{attribute 'monitoring' := 'variable'}
PROPERTY proAvailable : BOOL
GET
proAvailable := proIsReady;
END_GET
END_PROPERTY

{attribute 'monitoring' := 'variable'}
PROPERTY proLockDown : BOOL
GET
proLockDown := proIsError;
END_GET
END_PROPERTY

END_FUNCTION_BLOCK

// 21 Interface/ITF_SPERRANTRIEB
INTERFACE ITF_SPERRANTRIEB EXTENDS CtaAppBmk.ITF_BMK, CtaAppModbusSpezifikation.ITF_MODBUS_SPEZIFIKATION

PROPERTY proAuto : BOOL
GET
END_GET
SET
END_SET
END_PROPERTY

PROPERTY proHandOff : BOOL
GET
END_GET
SET
END_SET
END_PROPERTY

PROPERTY proHandOn : BOOL
GET
END_GET
SET
END_SET
END_PROPERTY

PROPERTY proIsRegulatet : BOOL
GET
END_GET
END_PROPERTY

PROPERTY proIsError : BOOL
GET
END_GET
END_PROPERTY

PROPERTY proIsWarning : BOOL
GET
END_GET
END_PROPERTY

PROPERTY proIsEnabled : BOOL
GET
END_GET
END_PROPERTY

PROPERTY proIsHandOnOrOff : BOOL
GET
END_GET
END_PROPERTY

PROPERTY proIsReady : BOOL
GET
END_GET
END_PROPERTY

PROPERTY proHardWareHandModulAktive : BOOL
GET
END_GET
END_PROPERTY

PROPERTY proRevisionSwitchOk : BOOL
GET
END_GET
END_PROPERTY

PROPERTY proHandManualClose : BOOL
SET
END_SET
GET
END_GET
END_PROPERTY

PROPERTY proEn : BOOL
SET
END_SET
GET
END_GET
END_PROPERTY

PROPERTY proRükIsOpen : BOOL
GET
END_GET
END_PROPERTY

PROPERTY proRükIsClosed : BOOL
GET
END_GET
END_PROPERTY

PROPERTY INTERNAL proStateSymbol : STRING
GET
END_GET
END_PROPERTY

PROPERTY INTERNAL proEnSymbol : STRING
GET
END_GET
END_PROPERTY

PROPERTY proOnZu : BOOL
GET
END_GET
END_PROPERTY

PROPERTY proIsOnY : REAL
GET
END_GET
END_PROPERTY

PROPERTY proOnAuf : BOOL
GET
END_GET
END_PROPERTY

PROPERTY proOnY : REAL
GET
END_GET
END_PROPERTY

PROPERTY proGetDI_RükIsOpen : BOOL
GET
END_GET
END_PROPERTY

PROPERTY proNotShowDI_RükIsOpen : BOOL
GET
END_GET
END_PROPERTY

PROPERTY proIsOpen_ITF : CtaSysIO.ITF_IO
GET
END_GET
END_PROPERTY

PROPERTY INTERNAL proGetDI_ActuatorHand : BOOL
GET
END_GET
END_PROPERTY

PROPERTY proNotShowDI_ActuatorHand : BOOL
GET
END_GET
END_PROPERTY

PROPERTY proHandModul_ITF : CtaSysIO.ITF_IO
GET
END_GET
END_PROPERTY

PROPERTY INTERNAL proGetDI_ActuatorFuseOk : BOOL
GET
END_GET
END_PROPERTY

PROPERTY proNotShowDI_ActuatorFuseOk : BOOL
GET
END_GET
END_PROPERTY

PROPERTY proActuatorFuse_ITF : CtaSysIO.ITF_IO
GET
END_GET
END_PROPERTY

PROPERTY INTERNAL proGetDI_IsReady : BOOL
GET
END_GET
END_PROPERTY

PROPERTY proNotShowDI_Ready : BOOL
GET
END_GET
END_PROPERTY

PROPERTY proActuatorReady_ITF : CtaSysIO.ITF_IO
GET
END_GET
END_PROPERTY

PROPERTY INTERNAL proGetDI_FuseOK : BOOL
GET
END_GET
END_PROPERTY

PROPERTY proNotShowDI_FuseOk : BOOL
GET
END_GET
END_PROPERTY

PROPERTY proFuse_ITF : CtaSysIO.ITF_IO
GET
END_GET
END_PROPERTY

PROPERTY INTERNAL proGetDI_RevisionSwitchOK : BOOL
GET
END_GET
END_PROPERTY

PROPERTY proNotShowDI_RevisionSwitchOk : BOOL
GET
END_GET
END_PROPERTY

PROPERTY proRevisionSwitch_ITF : CtaSysIO.ITF_IO
GET
END_GET
END_PROPERTY

PROPERTY proNotShowAI_ActualPosition : BOOL
GET
END_GET
END_PROPERTY

PROPERTY proGetAI_ActualPosition : REAL
GET
END_GET
END_PROPERTY

PROPERTY proActualPosition_ITF : CtaSysIO.ITF_IO
GET
END_GET
END_PROPERTY

PROPERTY proGetDI_RükIsClosed : BOOL
GET
END_GET
END_PROPERTY

PROPERTY proNotShowDI_RükIsClosed : BOOL
GET
END_GET
END_PROPERTY

PROPERTY proIsClosed_ITF : CtaSysIO.ITF_IO
GET
END_GET
END_PROPERTY

PROPERTY proOnY_ITF : CtaSysIO.ITF_IO
GET
END_GET
END_PROPERTY

PROPERTY proOnOpen_ITF : CtaSysIO.ITF_IO
GET
END_GET
END_PROPERTY

PROPERTY proOnClose_ITF : CtaSysIO.ITF_IO
GET
END_GET
END_PROPERTY

PROPERTY INTERNAL proAnzWarning : INT
GET
END_GET
END_PROPERTY

PROPERTY INTERNAL proITF_REPORTMANAGER : CtaAppReport.ITF_REPORTMANAGER
GET
END_GET
END_PROPERTY

PROPERTY INTERNAL proAnzInfo : INT
GET
END_GET
END_PROPERTY

PROPERTY INTERNAL proAnzError : INT
GET
END_GET
END_PROPERTY

PROPERTY INTERNAL proModbusTest : BOOL
SET
END_SET
GET
END_GET
END_PROPERTY

PROPERTY proModbusStateWord : REFERENCE TO ARRAY[0..3] OF WORD
GET
END_GET
END_PROPERTY

PROPERTY proModbusControllWord : REFERENCE TO ARRAY[0..3] OF WORD
GET
END_GET
END_PROPERTY

PROPERTY proConfigError : BOOL
GET
END_GET
END_PROPERTY

PROPERTY p_scBase_fbxEnable : CtaSysConfig.ITF_DATATYPE;
GET
END_GET
END_PROPERTY

PROPERTY p_scBase_fbxControllMb : CtaSysConfig.ITF_DATATYPE;
GET
END_GET
END_PROPERTY

PROPERTY p_scBase_fbxInvertiert : CtaSysConfig.ITF_DATATYPE;
GET
END_GET
END_PROPERTY

PROPERTY p_scBase_fbtSettingTime : CtaSysConfig.ITF_DATATYPE;
GET
END_GET
END_PROPERTY

PROPERTY p_scFuse_fbxEnable : CtaSysConfig.ITF_DATATYPE;
GET
END_GET
END_PROPERTY

PROPERTY p_scFuse_fbxInputMb : CtaSysConfig.ITF_DATATYPE;
GET
END_GET
END_PROPERTY

PROPERTY p_scFuse_fbxDoesAlarm : CtaSysConfig.ITF_DATATYPE;
GET
END_GET
END_PROPERTY

PROPERTY p_scActuatorFuse_fbxEnable : CtaSysConfig.ITF_DATATYPE;
GET
END_GET
END_PROPERTY

PROPERTY p_scActuatorFuse_fbxInputMb : CtaSysConfig.ITF_DATATYPE;
GET
END_GET
END_PROPERTY

PROPERTY p_scActuatorFuse_fbxDoesAlarm : CtaSysConfig.ITF_DATATYPE;
GET
END_GET
END_PROPERTY

PROPERTY p_scInSperrAtRevisionSwitch_fbxEnable : CtaSysConfig.ITF_DATATYPE;
GET
END_GET
END_PROPERTY

PROPERTY p_scInSperrAtRevisionSwitch_fbxInputMb : CtaSysConfig.ITF_DATATYPE;
GET
END_GET
END_PROPERTY

PROPERTY p_scInSperrAtReady_fbxEnable : CtaSysConfig.ITF_DATATYPE;
GET
END_GET
END_PROPERTY

PROPERTY p_scInSperrAtReady_fbxInputMb : CtaSysConfig.ITF_DATATYPE;
GET
END_GET
END_PROPERTY

PROPERTY p_scInSperrAtHand_fbxEnable : CtaSysConfig.ITF_DATATYPE;
GET
END_GET
END_PROPERTY

PROPERTY p_scInSperrAtHand_fbxInputMb : CtaSysConfig.ITF_DATATYPE;
GET
END_GET
END_PROPERTY

PROPERTY p_scInSperrAtRükClosed_fbxEnable : CtaSysConfig.ITF_DATATYPE;
GET
END_GET
END_PROPERTY

PROPERTY p_scInSperrAtRükClosed_fbxInputMb : CtaSysConfig.ITF_DATATYPE;
GET
END_GET
END_PROPERTY

PROPERTY p_scInSperrAtRükClosed_fbxDoesAlarm : CtaSysConfig.ITF_DATATYPE;
GET
END_GET
END_PROPERTY

PROPERTY p_scInSperrAtRükClosed_fbtDelayStart : CtaSysConfig.ITF_DATATYPE;
GET
END_GET
END_PROPERTY

PROPERTY p_scInSperrAtRükClosed_fbtDelayRun : CtaSysConfig.ITF_DATATYPE;
GET
END_GET
END_PROPERTY

PROPERTY p_scInSperrAtRükClosed_fbiTypeOfAck : CtaSysConfig.ITF_DATATYPE;
GET
END_GET
END_PROPERTY

PROPERTY p_scInSperrAtRükClosed_fbiMaxErrorRetryAllowed : CtaSysConfig.ITF_DATATYPE;
GET
END_GET
END_PROPERTY

PROPERTY p_scInSperrAtRükOpen_fbxEnable : CtaSysConfig.ITF_DATATYPE;
GET
END_GET
END_PROPERTY

PROPERTY p_scInSperrAtRükOpen_fbxInputMb : CtaSysConfig.ITF_DATATYPE;
GET
END_GET
END_PROPERTY

PROPERTY p_scInSperrAtRükOpen_fbxDoesAlarm : CtaSysConfig.ITF_DATATYPE;
GET
END_GET
END_PROPERTY

PROPERTY p_scInSperrAtRükOpen_fbtDelayStart : CtaSysConfig.ITF_DATATYPE;
GET
END_GET
END_PROPERTY

PROPERTY p_scInSperrAtRükOpen_fbtDelayRun : CtaSysConfig.ITF_DATATYPE;
GET
END_GET
END_PROPERTY

PROPERTY p_scInSperrAtRükOpen_fbiTypeOfAck : CtaSysConfig.ITF_DATATYPE;
GET
END_GET
END_PROPERTY

PROPERTY p_scInSperrAtRükOpen_fbiMaxErrorRetryAllowed : CtaSysConfig.ITF_DATATYPE;
GET
END_GET
END_PROPERTY

PROPERTY p_scInSperrAtActualPosition_fbxEnable : CtaSysConfig.ITF_DATATYPE;
GET
END_GET
END_PROPERTY

PROPERTY p_scInSperrAtActualPosition_fbxInputMb : CtaSysConfig.ITF_DATATYPE;
GET
END_GET
END_PROPERTY

PROPERTY p_scInSperrAtActualPosition_fbxDoesAlarm : CtaSysConfig.ITF_DATATYPE;
GET
END_GET
END_PROPERTY

PROPERTY p_scInSperrAtActualPosition_fbrMaxDiff : CtaSysConfig.ITF_DATATYPE;
GET
END_GET
END_PROPERTY

PROPERTY p_scInSperrAtActualPosition_fbtDelayStart : CtaSysConfig.ITF_DATATYPE;
GET
END_GET
END_PROPERTY

PROPERTY p_scInSperrAtActualPosition_fbtDelayRun : CtaSysConfig.ITF_DATATYPE;
GET
END_GET
END_PROPERTY

PROPERTY p_scInSperrAtActualPosition_fbiTypeOfAck : CtaSysConfig.ITF_DATATYPE;
GET
END_GET
END_PROPERTY

PROPERTY p_scInSperrAtActualPosition_fbiMaxErrorRetryAllowed : CtaSysConfig.ITF_DATATYPE;
GET
END_GET
END_PROPERTY

PROPERTY p_scInfluxDb_fbxEnable : CtaSysConfig.ITF_DATATYPE;
GET
END_GET
END_PROPERTY

PROPERTY p_scManual_fbxAlowManualOn : CtaSysConfig.ITF_DATATYPE;
GET
END_GET
END_PROPERTY

PROPERTY p_scManual_fbuiManualState : CtaSysConfig.ITF_DATATYPE;
GET
END_GET
END_PROPERTY

PROPERTY p_scManual_fbuiSchaltBefehl : CtaSysConfig.ITF_DATATYPE;
GET
END_GET
END_PROPERTY

PROPERTY proHandManualOpen : BOOL
GET
END_GET
SET
END_SET
END_PROPERTY

PROPERTY proIsInverted : BOOL
GET
END_GET
END_PROPERTY

PROPERTY proKlappenStatus : enKlappenStatus
GET
END_GET
END_PROPERTY

PROPERTY proValveIcon : UINT
GET
END_GET
SET
END_SET
END_PROPERTY

{attribute 'monitoring' := 'variable'}
PROPERTY proAcknowlege : BOOL
GET
END_GET
END_PROPERTY

{attribute 'monitoring' := 'variable'}
PROPERTY proAvailable : BOOL
GET
END_GET
END_PROPERTY

{attribute 'monitoring' := 'variable'}
PROPERTY proLockDown : BOOL
GET
END_GET
END_PROPERTY

PROPERTY proOn : BOOL
GET
END_GET
END_PROPERTY

END_INTERFACE

// 30 Program Organization Units/fcGetBigerStringValue
FUNCTION fcGetBigerStringValue : INT
VAR_INPUT
    st1     :   STRING(255);
    st2     :   STRING(255);
END_VAR
VAR
    diFor: DINT;
    diMax: DINT;
END_VAR

IF LEN(st1) > LEN(st2) THEN
    diMax := LEN(st2); 
    fcGetBigerStringValue := 1;
ELSIF LEN(st1) < LEN(st2) THEN
    diMax := LEN(st1);
    fcGetBigerStringValue := 2;     
ELSE
    diMax := LEN(st1);    
END_IF;
FOR diFor := 0 TO  diMax DO
    IF st1[diFor] > st2[diFor] THEN
        fcGetBigerStringValue := 1;  
        EXIT; 
    ELSIF st1[diFor] < st2[diFor] THEN
        fcGetBigerStringValue := 2;  
        EXIT;
    END_IF;
END_FOR;

END_FUNCTION

// 30 Program Organization Units/fcCheckQuerryReturnIcon
FUNCTION fcCheckQuerryReturnIcon : BOOL
VAR_INPUT
	_ITF_In			:	ITF_SPERRANTRIEB;
	_uiIconNr_In	:	UINT;
END_VAR

IF __QUERYINTERFACE(_ITF_In,_ITF_In) THEN	
	fcCheckQuerryReturnIcon := TRUE;	
	_ITF_In.proValveIcon := _uiIconNr_In;
ELSE
	fcCheckQuerryReturnIcon := FALSE;	
END_IF

END_FUNCTION

// 40 Visualizations/POPUP/SperrAntrieb_POPUP
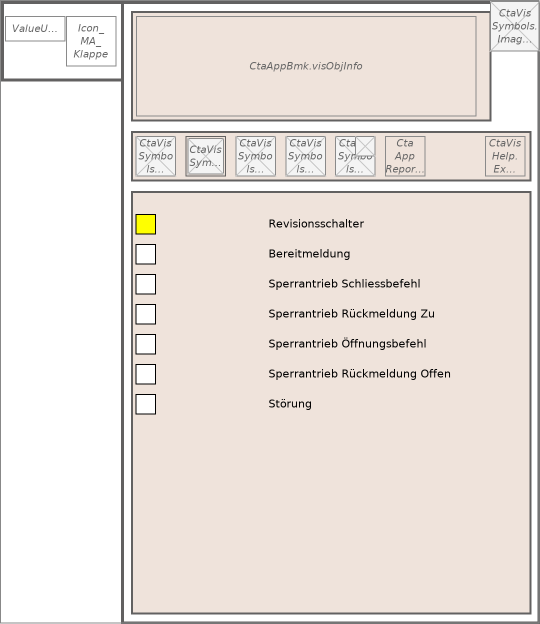
VISUALIZATION SperrAntrieb_POPUP  // 540x624
VAR_INPUT
    ITF_SPERRANTRIEBIN  :   ITF_SPERRANTRIEB;
    stExklParameter		:   STRING[40];	
	uiPopUpGruppe		: UINT;
END_VAR
    RoundedRectangle (1,1 160x80)
    RoundedRectangle (121,1 419x623)
    RoundedRectangle (131,11 360x110)
    RoundedRectangle (131,191 400x423)
    RoundedRectangle (131,131 400x50)
    Frame (136,16 340x100)
        shows CtaAppBmk.visObjInfo(ITF_BMK_IN := ITF_SPERRANTRIEBIN)
    Image (490,1 50x50), image: CtaVisSymbols.ImagePool.close_solo_black
        OnMouseClick:  Dialog=SperrAntrieb_POPUP, Result=None, NumpadKeypadSet=True
    Frame (131,204 399x400), frame switch variable: uiPopUpGruppe
        shows SperrAntrieb_OVERVIEW(ITF_SPERRANTRIEBIN := ITF_SPERRANTRIEBIN)
        shows SperrAntrieb_MANUAL(ITF_SPERRANTRIEBIN := ITF_SPERRANTRIEBIN)
        shows SperrAntrieb_PARAMETER(ITF_SPERRANTRIEBIN := ITF_SPERRANTRIEBIN)
        shows SperrAntrieb_IO(ITF_SPERRANTRIEBIN := ITF_SPERRANTRIEBIN)
        shows SperrAntrieb_BUS(ITF_SPERRANTRIEBIN := ITF_SPERRANTRIEBIN)
        shows SperrAntrieb_REPORTS(ITF_SPERRANTRIEBIN := ITF_SPERRANTRIEBIN)
        pReferences[2]: ITF_Parameter=ITF_SPERRANTRIEBIN.proParameter
    Frame (131,136 399x40)
        shows SperrAntrieb_PopUpListe(uiPopUpGruppe := uiPopUpGruppe, xHand := ITF_SPERRANTRIEBIN.proIsHandOnOrOff, xHandOff := ITF_SPERRANTRIEBIN.proHandOff, ITF_REPORTMANAGER_IN := ITF_SPERRANTRIEBIN.proITF_REPORTMANAGER, xBusTestAktiv := ITF_SPERRANTRIEBIN.proModbusTest, stExklParameter_IN := stExklParameter)
        pReferences[0]: AnzError=ITF_SPERRANTRIEBIN.proAnzError, AnzWarning=ITF_SPERRANTRIEBIN.proAnzWarning
    Frame (5,16 110x50), input disabled if: TRUE, frame switch variable: ITF_SPERRANTRIEBIN.proValveIcon
        shows SperrAntrieb_MA_Flap_Txt_L_Above(ITF_SPERRANTRIEB_IN := ITF_SPERRANTRIEBIN, stExklParameter := stExklParameter)
        shows SperrAntrieb_MB_Flap_Txt_L_Below(ITF_SPERRANTRIEB_IN := ITF_SPERRANTRIEBIN, stExklParameter := stExklParameter)
        shows SperrAntrieb_ML_Flap_Txt_L_Above(ITF_SPERRANTRIEB_IN := ITF_SPERRANTRIEBIN, stExklParameter := stExklParameter)
        shows SperrAntrieb_ML_Flap_Txt_L_Below(ITF_SPERRANTRIEB_IN := ITF_SPERRANTRIEBIN, stExklParameter := stExklParameter)
        shows SperrAntrieb_MA_Flap_Txt_R_Above(ITF_SPERRANTRIEB_IN := ITF_SPERRANTRIEBIN, stExklParameter := stExklParameter)
        shows SperrAntrieb_MB_Flap_Right_Txt_R_Below(ITF_SPERRANTRIEB_IN := ITF_SPERRANTRIEBIN, stExklParameter := stExklParameter)
        shows SperrAntrieb_MR_Flap_Txt_R_Above(ITF_SPERRANTRIEB_IN := ITF_SPERRANTRIEBIN, stExklParameter := stExklParameter)
        shows SperrAntrieb_MR_Flap_Txt_R_Below(ITF_SPERRANTRIEB_IN := ITF_SPERRANTRIEBIN, stExklParameter := stExklParameter)
        shows S_AT_ML_Valve_AB_Down_Txt_L_Above(ITF_STELLANTRIEB_IN := ITF_STELLANTRIEBIN)
        shows S_AT_ML_Valve_AB_Down_Txt_L_Below(ITF_STELLANTRIEB_IN := ITF_STELLANTRIEBIN)
        shows S_AT_ML_Valve_AB_Up_Txt_L_Above(ITF_STELLANTRIEB_IN := ITF_STELLANTRIEBIN)
        shows S_AT_ML_Valve_AB_Up_Txt_L_Below(ITF_STELLANTRIEB_IN := ITF_STELLANTRIEBIN)
        shows S_AT_ML_Valve_Flow_Txt_L_Above(ITF_STELLANTRIEB_IN := ITF_STELLANTRIEBIN)
        shows S_AT_ML_Valve_Flow_Txt_L_Below(ITF_STELLANTRIEB_IN := ITF_STELLANTRIEBIN)
        shows S_AT_ML_Valve_Mix_Txt_L_Above(ITF_STELLANTRIEB_IN := ITF_STELLANTRIEBIN)
        shows S_AT_ML_Valve_Mix_Txt_L_Below(ITF_STELLANTRIEB_IN := ITF_STELLANTRIEBIN)
        shows S_AT_MA_Valve_AB_Left_Txt_R_Above(ITF_STELLANTRIEB_IN := ITF_STELLANTRIEBIN)
        shows S_AT_MA_Valve_AB_Right_Txt_R_Above(ITF_STELLANTRIEB_IN := ITF_STELLANTRIEBIN)
        shows S_AT_MA_Valve_Flow_Txt_R_Above(ITF_STELLANTRIEB_IN := ITF_STELLANTRIEBIN)
        shows S_AT_MA_Valve_Mix_Txt_R_Above(ITF_STELLANTRIEB_IN := ITF_STELLANTRIEBIN)
        shows S_AT_MB_Valve_AB_Left_Txt_R_Below(ITF_STELLANTRIEB_IN := ITF_STELLANTRIEBIN)
        shows S_AT_MB_Valve_AB_Right_Txt_R_Below(ITF_STELLANTRIEB_IN := ITF_STELLANTRIEBIN)
        shows S_AT_MB_Valve_Flow_Txt_R_Below(ITF_STELLANTRIEB_IN := ITF_STELLANTRIEBIN)
        shows S_AT_MB_Valve_Mix_Txt_R_Below(ITF_STELLANTRIEB_IN := ITF_STELLANTRIEBIN)
        shows S_AT_MR_Valve_AB_Down_Txt_R_Above(ITF_STELLANTRIEB_IN := ITF_STELLANTRIEBIN)
        shows S_AT_MR_Valve_AB_Down_Txt_R_Below(ITF_STELLANTRIEB_IN := ITF_STELLANTRIEBIN)
        shows S_AT_MR_Valve_AB_Up_Txt_R_Above(ITF_STELLANTRIEB_IN := ITF_STELLANTRIEBIN)
        shows S_AT_MR_Valve_AB_Up_Txt_R_Below(ITF_STELLANTRIEB_IN := ITF_STELLANTRIEBIN)
        shows S_AT_MR_Valve_Flow_Txt_R_Above(ITF_STELLANTRIEB_IN := ITF_STELLANTRIEBIN)
        shows S_AT_MR_Valve_Flow_Txt_R_Below(ITF_STELLANTRIEB_IN := ITF_STELLANTRIEBIN)
        shows S_AT_MR_Valve_Mix_Txt_R_Above(ITF_STELLANTRIEB_IN := ITF_STELLANTRIEBIN)
        shows S_AT_MR_Valve_Mix_Txt_R_Below(ITF_STELLANTRIEB_IN := ITF_STELLANTRIEBIN)
        shows S_AT_MR_Valve_AB_Up_Txt_R_Above()
        shows S_AT_MR_Valve_AB_Up_Txt_R_Below()
        shows S_AT_MR_Flap_Txt_R_Above()
        shows S_AT_MR_Flap_Txt_R_Below()
        shows S_AT_MR_Valve_Flow_Txt_R_Above()
        shows S_AT_MR_Valve_Flow_Txt_R_Below()
        shows S_AT_MR_Valve_Mix_Txt_R_Above()
        shows S_AT_MR_Valve_Mix_Txt_R_Below()
END_VISUALIZATION

// 40 Visualizations/POPUP/SperrAntrieb_PopUpListe
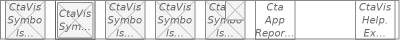
VISUALIZATION SperrAntrieb_PopUpListe  // 400x40
VAR_IN_OUT
	uiPopUpGruppe 			:	UINT;
END_VAR
VAR_INPUT
    xHand           		: 	BOOL;
    xHandOff        		: 	BOOL;
    ITF_REPORTMANAGER_IN 	: 	CtaAppReport.ITF_REPORTMANAGER;
    xBusTestAktiv   		: 	BOOL;	
	stExklParameter_IN		:	STRING[40];
END_VAR
    Group (5,0 40x40)
        RoundedRectangle (0,0 40x40), colour toggle: uiPopUpGruppe = 0
            OnMouseDown: execute { uiPopUpGruppe := 0; }
        Image (0,0 40x40), image: CtaVisSymbols.ImagePool.eye
            OnMouseDown: execute { uiPopUpGruppe := 0; }
    Group (105,0 40x40)
        RoundedRectangle (0,0 40x40), colour toggle: uiPopUpGruppe = 2
            OnMouseDown: execute { uiPopUpGruppe := 2; }
        Image (0,0 40x40), image: CtaVisSymbols.ImagePool.gear
            OnMouseDown: execute { uiPopUpGruppe := 2; }
    Group (55,0 40x40)
        RoundedRectangle (0,0 40x40), colour toggle: uiPopUpGruppe = 1
            OnMouseDown: execute { uiPopUpGruppe := 1; }
        Image (2,2 36x36), image: CtaVisSymbols.ImagePool.front_hand_Black
            OnMouseDown: execute { uiPopUpGruppe := 1; }
        Image (2,2 36x36), invisible if: NOT xHand, image: CtaVisSymbols.ImagePool.front_hand_Yellow
            OnMouseDown: execute { uiPopUpGruppe := 1; }
        Image (2,2 36x36), invisible if: NOT xHandOff, image: CtaVisSymbols.ImagePool.front_hand_Yellow_Off
            OnMouseDown: execute { uiPopUpGruppe := 1; }
    Group (155,0 40x40)
        RoundedRectangle (0,0 40x40), colour toggle: uiPopUpGruppe = 3
            OnMouseDown: execute { uiPopUpGruppe := 3; }
        Image (0,0 40x40), image: CtaVisSymbols.ImagePool.dip-switch
            OnMouseDown: execute { uiPopUpGruppe := 3; }
    Group (205,0 40x40)
        RoundedRectangle (0,0 40x40), colour toggle: uiPopUpGruppe = 4
            OnMouseDown: execute { uiPopUpGruppe := 4; }
        Image (0,0 40x40), image: CtaVisSymbols.ImagePool.lan
            OnMouseDown: execute { uiPopUpGruppe := 4; }
        Image (20,0 20x20), invisible if: NOT xBusTestAktiv, image: CtaVisSymbols.ImagePool.front_hand_Yellow
            OnMouseDown: execute { uiPopUpGruppe := 4; }
    Group (255,0 40x40)
        RoundedRectangle (0,0 40x40), colour toggle: uiPopUpGruppe = 5
            OnMouseDown: execute { uiPopUpGruppe := 5; }
        Frame (0,0 40x40), input disabled if: TRUE
            shows CtaAppReport.VIS_ANZ_REPORTS_MODUL(ITF_REPORTMANAGER_IN := ITF_REPORTMANAGER_IN)
            OnMouseDown: execute { uiPopUpGruppe := 5; }
    Group (355,0 40x40)
        RoundedRectangle (0,0 40x40), invisible if: stExklParameter_IN = ' '
        Frame (0,0 40x40)
            shows CtaVisHelp.ExkParameterSymbol(stExklParameter := stExklParameter_IN)
END_VISUALIZATION

// 40 Visualizations/ICON/SperrAntrieb_BASE/Icons/Motor
VISUALIZATION Motor  // 15x15
VAR_INPUT
    ITF_SPERRANTRIEB_IN   :   ITF_SPERRANTRIEB;	
END_VAR
    Ellipse (0,0 15x15), "M", colour toggle: ITF_SPERRANTRIEB_IN.proIsError
    Ellipse (0,0 15x15), "M", colour toggle: ITF_SPERRANTRIEB_IN.proOn, invisible if: ITF_SPERRANTRIEB_IN.proIsError
END_VISUALIZATION

// 40 Visualizations/POPUP/PARAMETER/SperrAntrieb_PARAMETER
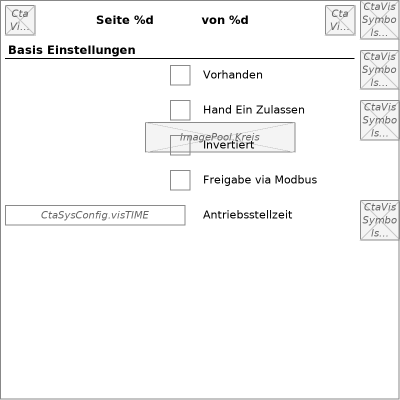
VISUALIZATION SperrAntrieb_PARAMETER  // 400x400
VAR_INPUT
    ITF_SPERRANTRIEBIN : ITF_SPERRANTRIEB;
END_VAR
VAR
    uiParameterGruppe : UINT;
END_VAR
    Image (145,122 150x30), image: ImagePool.Kreis
    Frame (360,0 40x300)
        shows SperrAntrieb_ParameterListe(uiParameterGruppe := uiParameterGruppe)
    Frame (0,0 360x400), frame switch variable: uiParameterGruppe
        shows SperrAntrieb_ParameterBase(ITF_SPERRANTRIEBIN := ITF_SPERRANTRIEBIN)
        shows SperrAntrieb_ParameterFuses(ITF_SPERRANTRIEBIN := ITF_SPERRANTRIEBIN)
        shows SperrAntrieb_ParameterIO(ITF_SPERRANTRIEBIN := ITF_SPERRANTRIEBIN)
        shows SperrAntrieb_ParameterInfluxDb(ITF_SPERRANTRIEBIN := ITF_SPERRANTRIEBIN)
        shows S_AT_ParameterInfluxDb(ITF_Parameter := ITF_Parameter)
        pReferences[0]: ITF_Parameter=ITF_Parameter
        pReferences[1]: ITF_Parameter=ITF_Parameter
        pReferences[2]: ITF_Parameter=ITF_Parameter
        pReferences[3]: ITF_Parameter=ITF_Parameter
END_VISUALIZATION

// 40 Visualizations/POPUP/PARAMETER/SperrAntrieb_ParameterListe
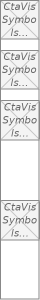
VISUALIZATION SperrAntrieb_ParameterListe  // 40x300
VAR_IN_OUT
	uiParameterGruppe : UINT;
END_VAR
    RoundedRectangle (0,100 39x39), colour toggle: uiParameterGruppe = 2
        OnMouseDown: execute { uiParameterGruppe := 2; }
    RoundedRectangle (0,50 39x39), colour toggle: uiParameterGruppe = 1
        OnMouseDown: execute { uiParameterGruppe := 1; }
    RoundedRectangle (0,0 39x39), colour toggle: uiParameterGruppe = 0
        OnMouseDown: execute { uiParameterGruppe := 0; }
    RoundedRectangle (0,200 39x39), colour toggle: uiParameterGruppe = 3
        OnMouseDown: execute { uiParameterGruppe := 3; }
    Image (0,0 39x39), image: CtaVisSymbols.ImagePool.valve_24dp_000000_FILL0_wght400_GRAD0_opsz24
        OnMouseDown: execute { uiParameterGruppe := 0; }
    Image (0,50 39x39), image: CtaVisSymbols.ImagePool.electric_bolt_24dp_000000_FILL0_wght400_GRAD0_opsz24
        OnMouseDown: execute { uiParameterGruppe := 1; }
    Image (0,100 40x40), image: CtaVisSymbols.ImagePool.dip-switch
        OnMouseDown: execute { uiParameterGruppe := 2; }
    Image (0,200 40x40), image: CtaVisSymbols.ImagePool.sine-wave
        OnMouseDown: execute { uiParameterGruppe := 3; }
END_VISUALIZATION

// 40 Visualizations/POPUP/MANUAL/SperrAntrieb_MANUAL
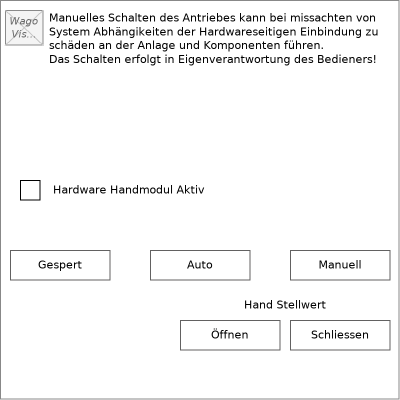
VISUALIZATION SperrAntrieb_MANUAL  // 400x400
VAR_INPUT
    ITF_SPERRANTRIEBIN    :   ITF_SPERRANTRIEB;	
END_VAR
    Label (46,10 350x100), "Manuelles Schalten des Antriebes kann bei missachten von System Abhängikeiten der Hardwareseitigen Einbindung zu schäden an der Anlage und Komponenten führen. Das Schalten erfolgt in Eigenverantwortung des Bedieners!"
    Image (5,10 38x35), image: WagoVisuIcons.WagoIcons.2
    Label (235,295 100x20), "Hand Stellwert"
    Rectangle (20,180 20x20), colour toggle: ITF_SPERRANTRIEBIN.proHardWareHandModulAktive, invisible if: NOT ITF_SPERRANTRIEBIN.proHardWareHandModulAktive
    Label (50,180 200x20), "Hardware Handmodul Aktiv", invisible if: NOT ITF_SPERRANTRIEBIN.proHardWareHandModulAktive
    RoundedRectangle (10,250 100x30), "Gespert", colour toggle: ITF_SPERRANTRIEBIN.proHandOff
        toggle ITF_SPERRANTRIEBIN.proHandOff
    RoundedRectangle (150,250 100x30), "Auto", colour toggle: ITF_SPERRANTRIEBIN.proAuto
        toggle ITF_SPERRANTRIEBIN.proAuto
    RoundedRectangle (290,250 100x30), "Manuell", colour toggle: ITF_SPERRANTRIEBIN.proHandOn
        toggle ITF_SPERRANTRIEBIN.proHandOn
    RoundedRectangle (180,320 100x30), "Öffnen", colour toggle: ITF_SPERRANTRIEBIN.proHandManualOpen, invisible if: NOT ITF_SPERRANTRIEBIN.proHandOn
        toggle ITF_SPERRANTRIEBIN.proHandManualOpen
    RoundedRectangle (290,320 100x30), "Schliessen", colour toggle: ITF_SPERRANTRIEBIN.proHandManualClose, invisible if: NOT ITF_SPERRANTRIEBIN.proHandOn
        toggle ITF_SPERRANTRIEBIN.proHandManualClose
END_VISUALIZATION

// 40 Visualizations/POPUP/OVERVIEW/SperrAntrieb_OVERVIEW
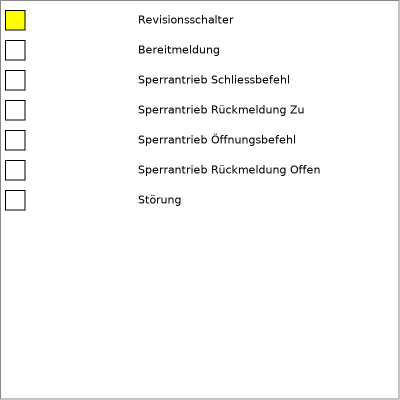
VISUALIZATION SperrAntrieb_OVERVIEW  // 400x400
VAR_INPUT
    ITF_SPERRANTRIEBIN    :   ITF_SPERRANTRIEB;	
END_VAR
    Label (135,10 250x20), "Revisionsschalter"
    Label (135,40 250x20), "Bereitmeldung"
    Rectangle (5,10 20x20), colour toggle: ITF_SPERRANTRIEBIN.proRevisionSwitchOk
    Rectangle (5,40 20x20), colour toggle: ITF_SPERRANTRIEBIN.proIsReady
    Rectangle (5,70 20x20), colour toggle: ITF_SPERRANTRIEBIN.proOnZu
    Label (135,70 250x20), "Sperrantrieb Schliessbefehl"
    Rectangle (5,100 20x20), colour toggle: ITF_SPERRANTRIEBIN.proRükIsClosed, invisible if: ITF_SPERRANTRIEBIN.proNotShowDI_RükIsClosed
    Label (135,100 250x20), "Sperrantrieb Rückmeldung Zu", invisible if: ITF_SPERRANTRIEBIN.proNotShowDI_RükIsClosed
    Rectangle (5,130 20x20), colour toggle: ITF_SPERRANTRIEBIN.proOnAuf
    Label (135,130 250x20), "Sperrantrieb Öffnungsbefehl"
    Rectangle (5,160 20x20), colour toggle: ITF_SPERRANTRIEBIN.proRükIsOpen, invisible if: ITF_SPERRANTRIEBIN.proNotShowDI_RükIsOpen
    Label (135,160 250x20), "Sperrantrieb Rückmeldung Offen", invisible if: ITF_SPERRANTRIEBIN.proNotShowDI_RükIsOpen
    Rectangle (5,190 20x20), colour toggle: ITF_SPERRANTRIEBIN.proIsError
    Label (135,190 250x20), "Störung"
END_VISUALIZATION

// 40 Visualizations/POPUP/BUS/SperrAntrieb_BUS
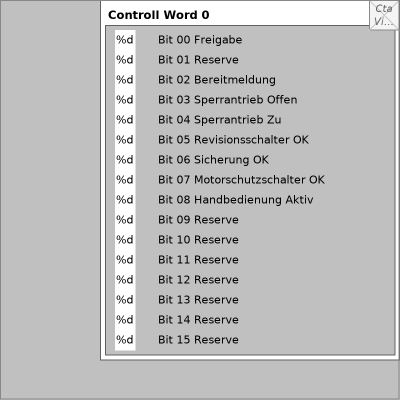
VISUALIZATION SperrAntrieb_BUS  // 400x400
VAR_INPUT
    ITF_SPERRANTRIEBIN    :   ITF_SPERRANTRIEB;	
END_VAR
    Frame (100,0 300x360)
        shows SperrAntrieb_BUS_CS(ITF_SPERRANTRIEBIn := ITF_SPERRANTRIEBIN, ayControllWord := ITF_SPERRANTRIEBIN.proModbusControllWord, ayStateWord := ITF_SPERRANTRIEBIN.proModbusStateWord)
END_VISUALIZATION

// 40 Visualizations/POPUP/BUS/SperrAntrieb_BUS_SW0_Detail
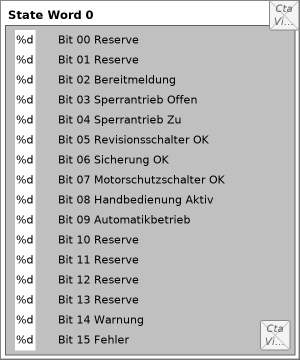
VISUALIZATION SperrAntrieb_BUS_SW0_Detail  // 300x360
VAR_IN_OUT
    wDetail     :   WORD;
END_VAR
VAR_INPUT	
    ITF_SPERRANTRIEBIN    :   ITF_SPERRANTRIEB;
END_VAR
VAR_IN_OUT
    xShow       :   BOOL;
END_VAR
    RoundedRectangle (0,0 300x360)
    RoundedRectangle (5,25 290x330)
    Textfield (15,30 20x20), "%d", text variable: TO_WORD(wDetail.0), input disabled if: NOT ITF_SPERRANTRIEBIn.proModbusTest
        OnMouseClick: execute { wDetail.0 := NOT wDetail.0; }
    Label (55,30 180x20), "Bit 00 Reserve"
    Textfield (15,50 20x20), "%d", text variable: TO_WORD(wDetail.1), input disabled if: NOT ITF_SPERRANTRIEBIn.proModbusTest
        OnMouseClick: execute { wDetail.1 := NOT wDetail.1; }
    Label (55,50 180x20), "Bit 01 Reserve"
    Textfield (15,70 20x20), "%d", text variable: TO_WORD(wDetail.2), input disabled if: NOT ITF_SPERRANTRIEBIn.proModbusTest
        OnMouseClick: execute { wDetail.2 := NOT wDetail.2; }
    Label (55,70 180x20), "Bit 02 Bereitmeldung"
    Textfield (15,90 20x20), "%d", text variable: TO_WORD(wDetail.3), input disabled if: NOT ITF_SPERRANTRIEBIn.proModbusTest
        OnMouseClick: execute { wDetail.3 := NOT wDetail.3; }
    Label (55,90 180x20), "Bit 03 Sperrantrieb Offen"
    Textfield (15,110 20x20), "%d", text variable: TO_WORD(wDetail.4), input disabled if: NOT ITF_SPERRANTRIEBIn.proModbusTest
        OnMouseClick: execute { wDetail.4 := NOT wDetail.4; }
    Label (55,110 180x20), "Bit 04 Sperrantrieb Zu"
    Textfield (15,130 20x20), "%d", text variable: TO_WORD(wDetail.5), input disabled if: NOT ITF_SPERRANTRIEBIn.proModbusTest
        OnMouseClick: execute { wDetail.5 := NOT wDetail.5; }
    Label (55,130 180x20), "Bit 05 Revisionsschalter OK"
    Textfield (15,150 20x20), "%d", text variable: TO_WORD(wDetail.6), input disabled if: NOT ITF_SPERRANTRIEBIn.proModbusTest
        OnMouseClick: execute { wDetail.6 := NOT wDetail.6; }
    Label (55,150 180x20), "Bit 06 Sicherung OK"
    Textfield (15,170 20x20), "%d", text variable: TO_WORD(wDetail.7), input disabled if: NOT ITF_SPERRANTRIEBIn.proModbusTest
        OnMouseClick: execute { wDetail.7 := NOT wDetail.7; }
    Label (55,170 180x20), "Bit 07 Motorschutzschalter OK"
    Textfield (15,190 20x20), "%d", text variable: TO_WORD(wDetail.8), input disabled if: NOT ITF_SPERRANTRIEBIn.proModbusTest
        OnMouseClick: execute { wDetail.8 := NOT wDetail.8; }
    Label (55,190 180x20), "Bit 08 Handbedienung Aktiv"
    Textfield (15,210 20x20), "%d", text variable: TO_WORD(wDetail.9), input disabled if: NOT ITF_SPERRANTRIEBIn.proModbusTest
        OnMouseClick: execute { wDetail.9 := NOT wDetail.9; }
    Label (55,210 180x20), "Bit 09 Automatikbetrieb"
    Textfield (15,230 20x20), "%d", text variable: TO_WORD(wDetail.10), input disabled if: NOT ITF_SPERRANTRIEBIn.proModbusTest
        OnMouseClick: execute { wDetail.10 := NOT wDetail.10; }
    Label (55,230 180x20), "Bit 10 Reserve"
    Textfield (15,250 20x20), "%d", text variable: TO_WORD(wDetail.11), input disabled if: NOT ITF_SPERRANTRIEBIn.proModbusTest
        OnMouseClick: execute { wDetail.11 := NOT wDetail.11; }
    Label (55,250 180x20), "Bit 11 Reserve"
    Textfield (15,270 20x20), "%d", text variable: TO_WORD(wDetail.12), input disabled if: NOT ITF_SPERRANTRIEBIn.proModbusTest
        OnMouseClick: execute { wDetail.12 := NOT wDetail.12; }
    Label (55,270 180x20), "Bit 12 Reserve"
    Textfield (15,290 20x20), "%d", text variable: TO_WORD(wDetail.13), input disabled if: NOT ITF_SPERRANTRIEBIn.proModbusTest
        OnMouseClick: execute { wDetail.13 := NOT wDetail.13; }
    Label (55,290 180x20), "Bit 13 Reserve"
    Textfield (15,310 20x20), "%d", text variable: TO_WORD(wDetail.14), input disabled if: NOT ITF_SPERRANTRIEBIn.proModbusTest
        OnMouseClick: execute { wDetail.14 := NOT wDetail.14; }
    Label (55,310 180x20), "Bit 14 Warnung"
    Textfield (15,330 20x20), "%d", text variable: TO_WORD(wDetail.15), input disabled if: NOT ITF_SPERRANTRIEBIn.proModbusTest
        OnMouseClick: execute { wDetail.15 := NOT wDetail.15; }
    Label (55,330 180x20), "Bit 15 Fehler"
    Label (5,0 150x30), "State Word 0"
    Image (260,320 30x30), invisible if: ITF_SPERRANTRIEBIN.proModbusTest, image: CtaVisSymbols.ImagePool.front_hand_Black
        OnMouseClick: execute { ITF_SPERRANTRIEBIN.proModbusTest := TRUE; }
    Image (260,320 30x30), invisible if: NOT ITF_SPERRANTRIEBIN.proModbusTest, image: CtaVisSymbols.ImagePool.front_hand_Yellow
        OnMouseClick: execute { ITF_SPERRANTRIEBIN.proModbusTest := False; }
    Image (269,0 30x30), image: CtaVisSymbols.ImagePool.close_solo_black
        OnMouseClick: execute { xShow := FALSE; ITF_SPERRANTRIEBIN.proModbusTest := FALSE; }
END_VISUALIZATION

// 40 Visualizations/POPUP/BUS/SperrAntrieb_BUS_CW0_Detail
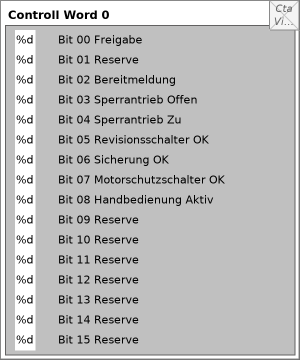
VISUALIZATION SperrAntrieb_BUS_CW0_Detail  // 300x360
VAR_IN_OUT
    wDetail :   WORD;
END_VAR
VAR_IN_OUT
    xShow   :   BOOL;
END_VAR
    RoundedRectangle (0,0 300x360)
    RoundedRectangle (5,25 290x330)
    Textfield (15,30 20x20), "%d", text variable: TO_WORD(wDetail.0), input disabled if: TRUE
    Label (55,30 180x20), "Bit 00 Freigabe"
    Textfield (15,50 20x20), "%d", text variable: TO_WORD(wDetail.1), input disabled if: TRUE
    Label (55,50 180x20), "Bit 01 Reserve"
    Textfield (15,70 20x20), "%d", text variable: TO_WORD(wDetail.2), input disabled if: TRUE
    Label (55,70 180x20), "Bit 02 Bereitmeldung"
    Textfield (15,90 20x20), "%d", text variable: TO_WORD(wDetail.3), input disabled if: TRUE
    Label (55,90 180x20), "Bit 03 Sperrantrieb Offen"
    Textfield (15,110 20x20), "%d", text variable: TO_WORD(wDetail.4), input disabled if: TRUE
    Label (55,110 180x20), "Bit 04 Sperrantrieb Zu"
    Textfield (15,130 20x20), "%d", text variable: TO_WORD(wDetail.5), input disabled if: TRUE
    Label (55,130 180x20), "Bit 05 Revisionsschalter OK"
    Textfield (15,150 20x20), "%d", text variable: TO_WORD(wDetail.6), input disabled if: TRUE
    Label (55,150 180x20), "Bit 06 Sicherung OK"
    Textfield (15,170 20x20), "%d", text variable: TO_WORD(wDetail.7), input disabled if: TRUE
    Label (55,170 180x20), "Bit 07 Motorschutzschalter OK"
    Textfield (15,190 20x20), "%d", text variable: TO_WORD(wDetail.8), input disabled if: TRUE
    Label (55,190 180x20), "Bit 08 Handbedienung Aktiv"
    Textfield (15,210 20x20), "%d", text variable: TO_WORD(wDetail.9), input disabled if: TRUE
    Label (55,210 180x20), "Bit 09 Reserve"
    Textfield (15,230 20x20), "%d", text variable: TO_WORD(wDetail.10), input disabled if: TRUE
    Label (55,230 180x20), "Bit 10 Reserve"
    Textfield (15,250 20x20), "%d", text variable: TO_WORD(wDetail.11), input disabled if: TRUE
    Label (55,250 180x20), "Bit 11 Reserve"
    Textfield (15,270 20x20), "%d", text variable: TO_WORD(wDetail.12), input disabled if: TRUE
    Label (55,270 180x20), "Bit 12 Reserve"
    Textfield (15,290 20x20), "%d", text variable: TO_WORD(wDetail.13), input disabled if: TRUE
    Label (55,290 180x20), "Bit 13 Reserve"
    Textfield (15,310 20x20), "%d", text variable: TO_WORD(wDetail.14), input disabled if: TRUE
    Label (55,310 180x20), "Bit 14 Reserve"
    Textfield (15,330 20x20), "%d", text variable: TO_WORD(wDetail.15), input disabled if: TRUE
    Label (55,330 180x20), "Bit 15 Reserve"
    Image (269,0 30x30), image: CtaVisSymbols.ImagePool.close_solo_black
        OnMouseClick: execute { xShow := FALSE; }
    Label (5,0 150x30), "Controll Word 0"
END_VISUALIZATION

// 40 Visualizations/POPUP/BUS/SperrAntrieb_BUS_CS
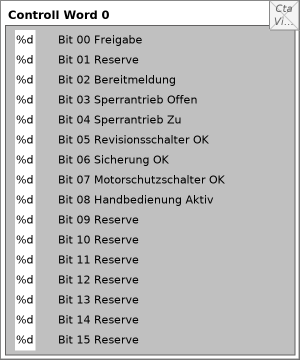
VISUALIZATION SperrAntrieb_BUS_CS  // 300x360
VAR_INPUT
    ITF_SPERRANTRIEBIn        :   ITF_SPERRANTRIEB;
    ayControllWord  :   REFERENCE TO ARRAY[0..3] OF WORD;
    ayStateWord     :   REFERENCE TO ARRAY[0..3] OF WORD;
END_VAR
VAR
    xShowCw :   BOOL;
    xShowSw :   BOOL;
    xShowSw1:   BOOL;
    xShowSw2:   BOOL;
END_VAR
    Textfield (0,10 130x20), "%b", text variable: ayControllWord[0]
    Label (140,10 120x20), "Controll Word 0"
    Label (140,50 120x20), "Controll Word 1"
    Textfield (0,50 130x20), "%d", text variable: ayControllWord[1]
    Label (140,90 120x20), "Controll Word 2", invisible if: TRUE
    Textfield (0,90 130x20), "%d", text variable: ayControllWord[2], invisible if: TRUE
    Label (140,130 120x20), "Controll Word 3", invisible if: TRUE
    Textfield (0,130 130x20), "%d", text variable: ayControllWord[3], invisible if: TRUE
    Image (265,5 30x30), image: CtaVisSymbols.ImagePool.information-variant
        OnMouseClick: execute {
            xShowCw := TRUE;
            xShowSw := FALSE;
            xShowSw1:= FALSE;
            xShowSw2:= FALSE;
        }
    Label (140,290 120x20), "State Word 3", invisible if: TRUE
    Textfield (0,170 130x20), "%b", text variable: ayStateWord[0]
        OnMouseDown: write the text variable via Default
    Label (140,170 120x20), "State Word 0"
    Label (140,210 120x20), "State Word 1"
    Textfield (0,210 130x20), "%d", text variable: ayStateWord[1]
    Label (140,250 120x20), "State Word 2"
    Textfield (0,250 130x20), "%d", text variable: ayStateWord[2]
    Textfield (0,290 130x20), "%d", text variable: ayStateWord[3], invisible if: TRUE
    Image (265,165 30x30), image: CtaVisSymbols.ImagePool.information-variant
        OnMouseClick: execute {
            xShowCw := FALSE;
            xShowSw := TRUE;
            xShowSw1:= FALSE;
            xShowSw2:= FALSE;
        }
    Image (265,205 30x30), image: CtaVisSymbols.ImagePool.information-variant
        OnMouseClick: execute {
            xShowCw := FALSE;
            xShowSw := FALSE;
            xShowSw1:= TRUE;
            xShowSw2:= FALSE;
        }
    Image (265,245 30x30), image: CtaVisSymbols.ImagePool.information-variant
        OnMouseClick: execute {
            xShowCw := FALSE;
            xShowSw := FALSE;
            xShowSw1:= FALSE;
            xShowSw2:= TRUE;
        }
    Frame (0,0 300x360), invisible if: NOT xShowSw
        shows SperrAntrieb_BUS_SW0_Detail(wDetail := ayStateWord[0], ITF_SPERRANTRIEBIN := ITF_SPERRANTRIEBIn, xShow := xShowSw)
    Frame (0,0 300x360), invisible if: NOT xShowSw1
        shows SperrAntrieb_BUS_SW1_Detail(wDetail := ayStateWord[1], ITF_SPERRANTRIEBIN := ITF_SPERRANTRIEBIn, xShow := xShowSw1)
    Frame (0,0 300x360), invisible if: NOT xShowSw2
        shows SperrAntrieb_BUS_SW2_Detail(wDetail := ayStateWord[2], ITF_SPERRANTRIEBIN := ITF_SPERRANTRIEBIn, xShow := xShowSw2)
        shows SperrAntrieb_BUS_SW2_Detail()
    Frame (0,0 300x360), invisible if: NOT xShowCw
        shows SperrAntrieb_BUS_CW0_Detail(wDetail := ayControllWord[0], xShow := xShowCw)
END_VISUALIZATION

// 40 Visualizations/POPUP/BUS/SperrAntrieb_BUS_SW1_Detail
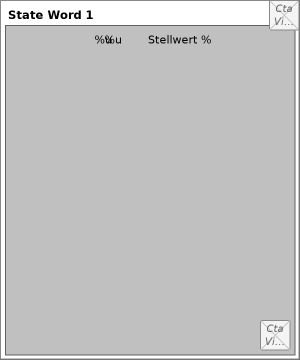
VISUALIZATION SperrAntrieb_BUS_SW1_Detail  // 300x360
VAR_IN_OUT
    wDetail     :   WORD;
END_VAR
VAR_INPUT	
    ITF_SPERRANTRIEBIN    :   ITF_SPERRANTRIEB;
END_VAR
VAR_IN_OUT
    xShow       :   BOOL;
END_VAR
    RoundedRectangle (0,0 300x360)
    RoundedRectangle (5,25 290x330)
    Image (269,0 30x30), image: CtaVisSymbols.ImagePool.close_solo_black
        OnMouseClick: execute { xShow := FALSE; ITF_SPERRANTRIEBIN.proModbusTest := FALSE; }
    Label (5,0 150x30), "State Word 1"
    Label (145,30 120x20), "Stellwert %"
    Textfield (5,30 110x20), "%u", text variable: wDetail, input disabled if: NOT ITF_SPERRANTRIEBIn.proModbusTest
        OnMouseClick: write the text variable via InputWithLimits, min 0, max 100
    Textfield (15,30 110x20), "%u", text variable: wDetail, invisible if: ITF_SPERRANTRIEBIN.proModbusTest
    Image (260,320 30x30), invisible if: ITF_SPERRANTRIEBIN.proModbusTest, image: CtaVisSymbols.ImagePool.front_hand_Black
        OnMouseClick: execute { ITF_SPERRANTRIEBIN.proModbusTest := TRUE; }
    Image (260,320 30x30), invisible if: NOT ITF_SPERRANTRIEBIN.proModbusTest, image: CtaVisSymbols.ImagePool.front_hand_Yellow
        OnMouseClick: execute { ITF_SPERRANTRIEBIN.proModbusTest := False; }
END_VISUALIZATION

// 40 Visualizations/POPUP/BUS/SperrAntrieb_BUS_SW2_Detail
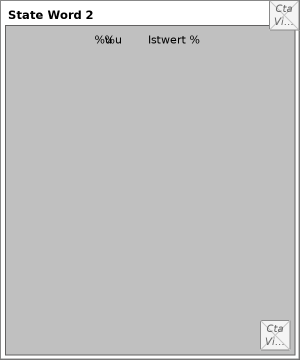
VISUALIZATION SperrAntrieb_BUS_SW2_Detail  // 300x360
VAR_IN_OUT
    wDetail             :   WORD;
END_VAR
VAR_INPUT	
    ITF_SPERRANTRIEBIN       :   ITF_SPERRANTRIEB;
END_VAR
VAR_IN_OUT
    xShow               :   BOOL;
END_VAR
    RoundedRectangle (0,0 300x360)
    RoundedRectangle (5,25 290x330)
    Image (269,0 30x30), image: CtaVisSymbols.ImagePool.close_solo_black
        OnMouseClick: execute { xShow := FALSE; ITF_SPERRANTRIEBIN.proModbusTest := FALSE; }
    Label (5,0 150x30), "State Word 2"
    Label (145,30 120x20), "Istwert %"
    Textfield (5,30 110x20), "%u", text variable: wDetail, input disabled if: NOT ITF_SPERRANTRIEBIn.proModbusTest
        OnMouseClick: write the text variable via InputWithLimits, min 0, max 100
    Textfield (15,30 110x20), "%u", text variable: wDetail, invisible if: ITF_SPERRANTRIEBIN.proModbusTest
    Image (260,320 30x30), invisible if: ITF_SPERRANTRIEBIN.proModbusTest, image: CtaVisSymbols.ImagePool.front_hand_Black
        OnMouseClick: execute { ITF_SPERRANTRIEBIN.proModbusTest := TRUE; }
    Image (260,320 30x30), invisible if: NOT ITF_SPERRANTRIEBIN.proModbusTest, image: CtaVisSymbols.ImagePool.front_hand_Yellow
        OnMouseClick: execute { ITF_SPERRANTRIEBIN.proModbusTest := False; }
END_VISUALIZATION

// 40 Visualizations/POPUP/REPORTS/SperrAntrieb_REPORTS
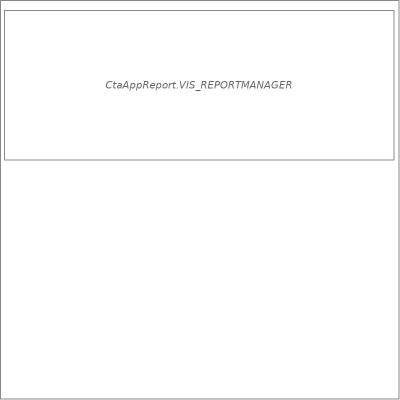
VISUALIZATION SperrAntrieb_REPORTS  // 400x400
VAR_INPUT
    ITF_SPERRANTRIEBIN    :   ITF_SPERRANTRIEB;	
END_VAR
    Frame (4,10 390x150)
        shows CtaAppReport.VIS_REPORTMANAGER(ITF_REPORTMANAGER := ITF_SPERRANTRIEBIN.proITF_REPORTMANAGER)
END_VISUALIZATION

// 40 Visualizations/POPUP/PARAMETER/SperrAntrieb_ParameterBase/SperrAntrieb_ParameterBase0
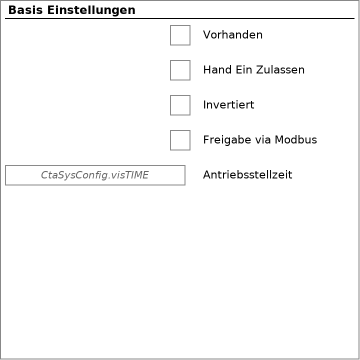
VISUALIZATION SperrAntrieb_ParameterBase0  // 360x360
VAR_INPUT
    ITF_SPERRANTRIEBIN : ITF_SPERRANTRIEB;
END_VAR
    Label (5,0 350x20), "Basis Einstellungen"
    Frame (170,25 20x20)
        shows CtaSysConfig.visBOOL(visfbBOOLIn := ITF_SPERRANTRIEBIN.p_scBase_fbxEnable)
    Label (200,25 150x20), "Vorhanden"
    Label (200,130 150x20), "Freigabe via Modbus"
    Frame (170,130 20x20)
        shows CtaSysConfig.visBOOL(visfbBOOLIn := ITF_SPERRANTRIEBIN.p_scBase_fbxControllMb)
    Frame (170,60 20x20)
        shows CtaSysConfig.visBOOL(visfbBOOLIn := ITF_SPERRANTRIEBIN.p_scManual_fbxAlowManualOn)
    Label (200,60 150x20), "Hand Ein Zulassen"
    Frame (170,95 20x20)
        shows CtaSysConfig.visBOOL(visfbBOOLIn := ITF_SPERRANTRIEBIN.p_scBase_fbxInvertiert)
    Label (200,95 150x20), "Invertiert"
    Label (200,165 150x20), "Antriebsstellzeit"
    Frame (5,165 180x20)
        shows CtaSysConfig.visTIME(visfbTIMEIn := ITF_SPERRANTRIEBIN.p_scBase_fbtSettingTime)
    Line (5,18) (354,18)
END_VISUALIZATION

// 40 Visualizations/POPUP/PARAMETER/SperrAntrieb_ParameterBase/SperrAntrieb_ParameterBase
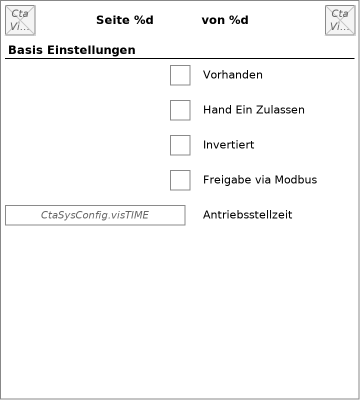
VISUALIZATION SperrAntrieb_ParameterBase  // 360x400
VAR_INPUT
    ITF_SPERRANTRIEBIN : ITF_SPERRANTRIEB;
END_VAR
VAR
    uiPage  :   UINT;
    uiMin   :   UINT    := 0;
    uiMax   :   UINT    := 0;
END_VAR
    Image (5,5 30x30), invisible if: uiPage = uiMin, image: CtaVisSymbols.ImagePool.arrow-left_square
        OnMouseClick: execute {
            uiPage := uiPage - 1;
            IF uiPage <= uiMin THEN
                uiPage := uiMin;
            END_IF;
        }
    Image (325,5 30x30), invisible if: uiPage = uiMax, image: CtaVisSymbols.ImagePool.arrow-right_square
        OnMouseClick: execute {
            uiPage := uiPage + 1;
            IF uiPage >= uiMax THEN
                uiPage := uiMax;
            END_IF;
        }
    Frame (0,40 360x360), frame switch variable: uiPage
        shows SperrAntrieb_ParameterBase0(ITF_SPERRANTRIEBIN := ITF_SPERRANTRIEBIN)
        shows S_AT_ParameterBase1()
        shows S_AT_ParameterBase3()
        shows SperrAT_ParameterBase1(ITF_Parameter := ITF_Parameter)
        pReferences[0]: ITF_Parameter=ITF_Parameter
        p982447995: ITF_Parameter
        p2498127594: ITF_Parameter
    Textfield (175,5 100x30), "von %d", text variable: uiMax
    Textfield (75,5 100x30), "Seite %d", text variable: uiPage
END_VISUALIZATION

// 40 Visualizations/POPUP/PARAMETER/SperrAntrieb_Fuse/SperrAntrieb_ParameterFuses0
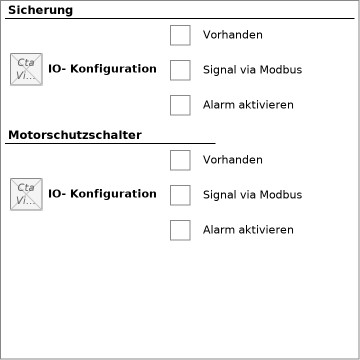
VISUALIZATION SperrAntrieb_ParameterFuses0  // 360x360
VAR_INPUT
    ITF_SPERRANTRIEBIN 	:	ITF_SPERRANTRIEB;
	ITF_Fuse_IN 		:	CtaSysIO.ITF_IO;
	ITF_ActuatorFuse_IN :	CtaSysIO.ITF_IO;
END_VAR
    Frame (170,25 20x20)
        shows CtaSysConfig.visBOOL(visfbBOOLIn := ITF_SPERRANTRIEBIN.p_scFuse_fbxEnable)
    Label (200,25 150x20), "Vorhanden"
    Frame (170,60 20x20)
        shows CtaSysConfig.visBOOL(visfbBOOLIn := ITF_SPERRANTRIEBIN.p_scFuse_fbxInputMb)
    Label (200,60 150x20), "Signal via Modbus"
    Frame (170,95 20x20)
        shows CtaSysConfig.visBOOL(visfbBOOLIn := ITF_SPERRANTRIEBIN.p_scFuse_fbxDoesAlarm)
    Label (200,95 150x20), "Alarm aktivieren"
    Label (5,0 350x20), "Sicherung"
    Label (5,125 350x20), "Motorschutzschalter"
    Frame (170,150 20x20)
        shows CtaSysConfig.visBOOL(visfbBOOLIn := ITF_SPERRANTRIEBIN.p_scActuatorFuse_fbxEnable)
    Label (200,150 150x20), "Vorhanden"
    Frame (170,185 20x20)
        shows CtaSysConfig.visBOOL(visfbBOOLIn := ITF_SPERRANTRIEBIN.p_scActuatorFuse_fbxInputMb)
    Label (200,185 150x20), "Signal via Modbus"
    Frame (170,220 20x20)
        shows CtaSysConfig.visBOOL(visfbBOOLIn := ITF_SPERRANTRIEBIN.p_scActuatorFuse_fbxDoesAlarm)
    Label (200,220 150x20), "Alarm aktivieren"
    Line (5,143) (215,143)
    Line (5,18) (354,18)
    Image (10,53 32x32), invisible if: ITF_Fuse_IN = 0, image: CtaVisSymbols.ImagePool.build
        OnMouseDown:  Dialog=SperrAntrieb_POPUP_IO_ITF, Parameters={ITF_IO_IN: ITF_Fuse_IN}, OpenModal=True, OpenCentered=True
    Label (45,59 120x20), "IO- Konfiguration", invisible if: ITF_Fuse_IN = 0
    Image (10,178 32x32), invisible if: ITF_ActuatorFuse_IN = 0, image: CtaVisSymbols.ImagePool.build
        OnMouseDown:  Dialog=SperrAntrieb_POPUP_IO_ITF, Parameters={ITF_IO_IN: ITF_ActuatorFuse_IN}, OpenModal=True, OpenCentered=True
    Label (45,184 120x20), "IO- Konfiguration", invisible if: ITF_ActuatorFuse_IN = 0
END_VISUALIZATION

// 40 Visualizations/POPUP/PARAMETER/SperrAntrieb_Fuse/SperrAntrieb_ParameterFuses
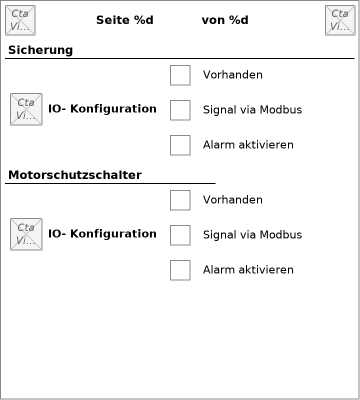
VISUALIZATION SperrAntrieb_ParameterFuses  // 360x400
VAR_INPUT
    ITF_SPERRANTRIEBIN : ITF_SPERRANTRIEB;
END_VAR
VAR
    uiPage  :   UINT;
    uiMin   :   UINT    := 0;
    uiMax   :   UINT    := 0;
END_VAR
    Image (5,5 30x30), invisible if: uiPage = uiMin, image: CtaVisSymbols.ImagePool.arrow-left_square
        OnMouseClick: execute {
            uiPage := uiPage - 1;
            IF uiPage <= uiMin THEN
                uiPage := uiMin;
            END_IF;
        }
    Image (325,5 30x30), invisible if: uiPage = uiMax, image: CtaVisSymbols.ImagePool.arrow-right_square
        OnMouseClick: execute {
            uiPage := uiPage + 1;
            IF uiPage >= uiMax THEN
                uiPage := uiMax;
            END_IF;
        }
    Frame (0,40 360x360), frame switch variable: uiPage
        shows SperrAntrieb_ParameterFuses0(ITF_SPERRANTRIEBIN := ITF_SPERRANTRIEBIN, ITF_Fuse_IN := ITF_SPERRANTRIEBIN.proFuse_ITF, ITF_ActuatorFuse_IN := ITF_SPERRANTRIEBIN.proActuatorFuse_ITF)
        shows AT_ParameterIO1(ITF_Parameter := ITF_Parameter)
        pReferences[0]: ITF_Parameter=ITF_Parameter
    Textfield (75,5 100x30), "Seite %d", text variable: uiPage
    Textfield (175,5 100x30), "von %d", text variable: uiMax
END_VISUALIZATION

// 40 Visualizations/POPUP/PARAMETER/SperrAntrieb_IO/SperrAntrieb_ParameterIO0
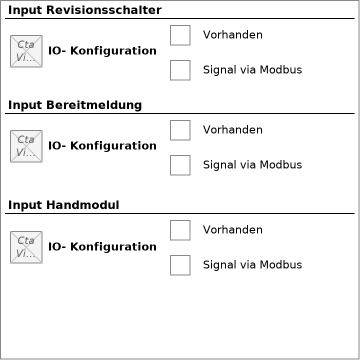
VISUALIZATION SperrAntrieb_ParameterIO0  // 360x360
VAR_INPUT
    ITF_SPERRANTRIEBIN 	:	ITF_SPERRANTRIEB;
	ITF_RevSwitch_IN 	:	CtaSysIO.ITF_IO;
	ITF_Ready_IN 		:	CtaSysIO.ITF_IO;
	ITF_HandModul_IN 	:	CtaSysIO.ITF_IO;
END_VAR
    Frame (170,25 20x20)
        shows CtaSysConfig.visBOOL(visfbBOOLIn := ITF_SPERRANTRIEBIN.p_scInSperrAtRevisionSwitch_fbxEnable)
    Label (200,25 150x20), "Vorhanden"
    Frame (170,60 20x20)
        shows CtaSysConfig.visBOOL(visfbBOOLIn := ITF_SPERRANTRIEBIN.p_scInSperrAtRevisionSwitch_fbxInputMb)
    Label (200,60 150x20), "Signal via Modbus"
    Label (5,0 350x20), "Input Revisionsschalter"
    Label (5,95 350x20), "Input Bereitmeldung"
    Frame (170,120 20x20)
        shows CtaSysConfig.visBOOL(visfbBOOLIn := ITF_SPERRANTRIEBIN.p_scInSperrAtReady_fbxEnable)
    Label (200,120 150x20), "Vorhanden"
    Frame (170,155 20x20)
        shows CtaSysConfig.visBOOL(visfbBOOLIn := ITF_SPERRANTRIEBIN.p_scInSperrAtReady_fbxInputMb)
    Label (200,155 150x20), "Signal via Modbus"
    Label (5,195 350x20), "Input Handmodul"
    Frame (170,220 20x20)
        shows CtaSysConfig.visBOOL(visfbBOOLIn := ITF_SPERRANTRIEBIN.p_scInSperrAtHand_fbxEnable)
    Label (200,220 150x20), "Vorhanden"
    Frame (170,255 20x20)
        shows CtaSysConfig.visBOOL(visfbBOOLIn := ITF_SPERRANTRIEBIN.p_scInSperrAtHand_fbxInputMb)
    Label (200,255 150x20), "Signal via Modbus"
    Line (5,18) (354,18)
    Line (5,113) (354,113)
    Line (5,213) (354,213)
    Image (10,231 32x32), invisible if: ITF_HandModul_IN = 0, image: CtaVisSymbols.ImagePool.build
        OnMouseDown:  Dialog=SperrAntrieb_POPUP_IO_ITF, Parameters={ITF_IO_IN: ITF_HandModul_IN}, OpenModal=True, OpenCentered=True
    Image (10,35 32x32), invisible if: ITF_RevSwitch_IN = 0, image: CtaVisSymbols.ImagePool.build
        OnMouseDown:  Dialog=SperrAntrieb_POPUP_IO_ITF, Parameters={ITF_IO_IN: ITF_RevSwitch_IN}, OpenModal=True, OpenCentered=True
    Label (45,41 120x20), "IO- Konfiguration", invisible if: ITF_RevSwitch_IN = 0
    Image (10,130 32x32), invisible if: ITF_Ready_IN = 0, image: CtaVisSymbols.ImagePool.build
        OnMouseDown:  Dialog=SperrAntrieb_POPUP_IO_ITF, Parameters={ITF_IO_IN: ITF_Ready_IN}, OpenModal=True, OpenCentered=True
    Label (45,136 120x20), "IO- Konfiguration", invisible if: ITF_Ready_IN = 0
    Label (45,237 120x20), "IO- Konfiguration", invisible if: ITF_HandModul_IN = 0
END_VISUALIZATION

// 40 Visualizations/POPUP/PARAMETER/SperrAntrieb_IO/SperrAntrieb_ParameterIO1
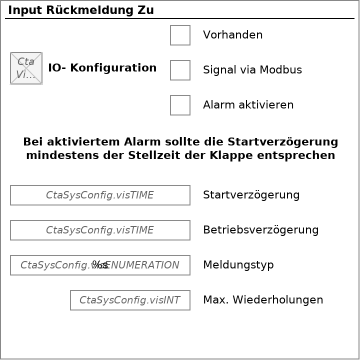
VISUALIZATION SperrAntrieb_ParameterIO1  // 360x360
VAR_INPUT
    ITF_SPERRANTRIEBIN 	:	ITF_SPERRANTRIEB;
	ITF_RückClosed_IN	:	CtaSysIO.ITF_IO;
END_VAR
    Label (5,0 350x20), "Input Rückmeldung Zu"
    Frame (170,25 20x20)
        shows CtaSysConfig.visBOOL(visfbBOOLIn := ITF_SPERRANTRIEBIN.p_scInSperrAtRükClosed_fbxEnable)
    Label (200,25 150x20), "Vorhanden"
    Frame (170,60 20x20)
        shows CtaSysConfig.visBOOL(visfbBOOLIn := ITF_SPERRANTRIEBIN.p_scInSperrAtRükClosed_fbxInputMb)
    Label (200,60 150x20), "Signal via Modbus"
    Frame (170,95 20x20)
        shows CtaSysConfig.visBOOL(visfbBOOLIn := ITF_SPERRANTRIEBIN.p_scInSperrAtRükClosed_fbxDoesAlarm)
    Label (200,95 150x20), "Alarm aktivieren"
    Frame (10,185 180x20)
        shows CtaSysConfig.visTIME(visfbTIMEIn := ITF_SPERRANTRIEBIN.p_scInSperrAtRükClosed_fbtDelayStart)
    Label (200,185 150x20), "Startverzögerung"
    Label (200,220 150x20), "Betriebsverzögerung"
    Frame (10,220 180x20)
        shows CtaSysConfig.visTIME(visfbTIMEIn := ITF_SPERRANTRIEBIN.p_scInSperrAtRükClosed_fbtDelayRun)
    Label (5,135 352x27), "Bei aktiviertem Alarm sollte die Startverzögerung mindestens der Stellzeit der Klappe entsprechen"
    Label (200,255 150x20), "Meldungstyp"
    Label (200,290 150x20), "Max. Wiederholungen"
    Line (5,18) (354,18)
    Frame (10,255 180x20)
        shows CtaSysConfig.visENUMERATION(visfbENUIn := ITF_SPERRANTRIEBIN.p_scInSperrAtRükClosed_fbiTypeOfAck)
    Frame (70,290 120x20)
        shows CtaSysConfig.visINT(visfbINTIn := ITF_SPERRANTRIEBIN.p_scInSperrAtRükClosed_fbiMaxErrorRetryAllowed)
    Image (10,52 32x32), invisible if: ITF_RückClosed_IN = 0, image: CtaVisSymbols.ImagePool.build
        OnMouseDown:  Dialog=SperrAntrieb_POPUP_IO_ITF, Parameters={ITF_IO_IN: ITF_RückClosed_IN}, OpenModal=True, OpenCentered=True
    Label (45,58 120x20), "IO- Konfiguration", invisible if: ITF_RückClosed_IN = 0
    Textfield (30,255 140x20), "%s", text list: 'CtaAppReport.txtLibAp99_2enTypeOfAck', text index: CtaSysConfig.fcGetEnumerationId(ITF_SPERRANTRIEBIN.p_scInSperrAtRükClosed_fbiTypeOfAck)
END_VISUALIZATION

// 40 Visualizations/POPUP/PARAMETER/SperrAntrieb_IO/SperrAntrieb_ParameterIO
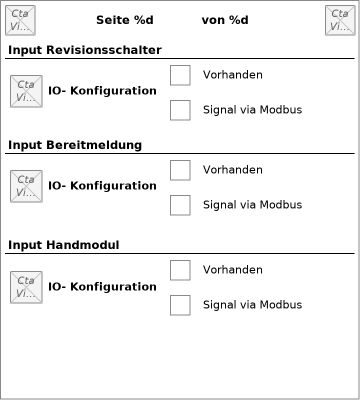
VISUALIZATION SperrAntrieb_ParameterIO  // 360x400
VAR_INPUT
    ITF_SPERRANTRIEBIN : ITF_SPERRANTRIEB;
END_VAR
VAR
    uiPage  :   UINT;
    uiMin   :   UINT    := 0;
    uiMax   :   UINT    := 4;
END_VAR
    Frame (0,40 360x360), frame switch variable: uiPage
        shows SperrAntrieb_ParameterIO0(ITF_SPERRANTRIEBIN := ITF_SPERRANTRIEBIN, ITF_RevSwitch_IN := ITF_SPERRANTRIEBIN.proRevisionSwitch_ITF, ITF_Ready_IN := ITF_SPERRANTRIEBIN.proActuatorReady_ITF, ITF_HandModul_IN := ITF_SPERRANTRIEBIN.proHandModul_ITF)
        shows SperrAntrieb_ParameterIO1(ITF_SPERRANTRIEBIN := ITF_SPERRANTRIEBIN, ITF_RückClosed_IN := ITF_SPERRANTRIEBIN.proIsClosed_ITF)
        shows SperrAntrieb_ParameterIO2(ITF_SPERRANTRIEBIN := ITF_SPERRANTRIEBIN, ITF_RückOffen_IN := ITF_SPERRANTRIEBIN.proIsOpen_ITF)
        shows SperrAntrieb_ParameterIO3(ITF_SPERRANTRIEBIN := ITF_SPERRANTRIEBIN, ITF_ActualPos_IN := ITF_SPERRANTRIEBIN.proActualPosition_ITF)
        shows SperrAntrieb_ParameterIO4(ITF_SPERRANTRIEBIN := ITF_SPERRANTRIEBIN, ITF_xOnAuf_IN := ITF_SPERRANTRIEBIN.proOnOpen_ITF, ITF_xOnZu_IN := ITF_SPERRANTRIEBIN.proOnClose_ITF, ITF_rOnY_IN := ITF_SPERRANTRIEBIN.proOnY_ITF)
    Image (325,5 30x30), invisible if: uiPage = uiMax, image: CtaVisSymbols.ImagePool.arrow-right_square
        OnMouseClick: execute {
            uiPage := uiPage + 1;
            IF uiPage >= uiMax THEN
                uiPage := uiMax;
            END_IF;
        }
    Image (5,5 30x30), invisible if: uiPage = uiMin, image: CtaVisSymbols.ImagePool.arrow-left_square
        OnMouseClick: execute {
            uiPage := uiPage - 1;
            IF uiPage <= uiMin THEN
                uiPage := uiMin;
            END_IF;
        }
    Textfield (175,5 100x30), "von %d", text variable: uiMax
    Textfield (75,5 100x30), "Seite %d", text variable: uiPage
END_VISUALIZATION

// 40 Visualizations/POPUP/PARAMETER/SperrAntrieb_IO/SperrAntrieb_ParameterIO2
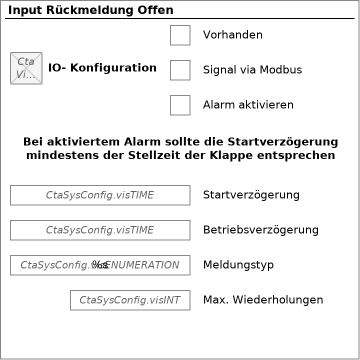
VISUALIZATION SperrAntrieb_ParameterIO2  // 360x360
VAR_INPUT
    ITF_SPERRANTRIEBIN 	:	ITF_SPERRANTRIEB;
	ITF_RückOffen_IN	:	CtaSysIO.ITF_IO;
END_VAR
    Label (5,0 350x20), "Input Rückmeldung Offen"
    Frame (170,25 20x20)
        shows CtaSysConfig.visBOOL(visfbBOOLIn := ITF_SPERRANTRIEBIN.p_scInSperrAtRükOpen_fbxEnable)
    Label (200,25 150x20), "Vorhanden"
    Frame (170,60 20x20)
        shows CtaSysConfig.visBOOL(visfbBOOLIn := ITF_SPERRANTRIEBIN.p_scInSperrAtRükOpen_fbxInputMb)
    Label (200,60 150x20), "Signal via Modbus"
    Frame (170,95 20x20)
        shows CtaSysConfig.visBOOL(visfbBOOLIn := ITF_SPERRANTRIEBIN.p_scInSperrAtRükOpen_fbxDoesAlarm)
    Label (200,95 150x20), "Alarm aktivieren"
    Frame (10,185 180x20)
        shows CtaSysConfig.visTIME(visfbTIMEIn := ITF_SPERRANTRIEBIN.p_scInSperrAtRükOpen_fbtDelayStart)
    Label (200,185 150x20), "Startverzögerung"
    Label (200,220 150x20), "Betriebsverzögerung"
    Frame (10,220 180x20)
        shows CtaSysConfig.visTIME(visfbTIMEIn := ITF_SPERRANTRIEBIN.p_scInSperrAtRükOpen_fbtDelayRun)
    Label (5,135 352x27), "Bei aktiviertem Alarm sollte die Startverzögerung mindestens der Stellzeit der Klappe entsprechen"
    Label (200,255 150x20), "Meldungstyp"
    Label (200,290 150x20), "Max. Wiederholungen"
    Line (5,18) (354,18)
    Frame (10,255 180x20)
        shows CtaSysConfig.visENUMERATION(visfbENUIn := ITF_SPERRANTRIEBIN.p_scInSperrAtRükOpen_fbiTypeOfAck)
    Frame (70,290 120x20)
        shows CtaSysConfig.visINT(visfbINTIn := ITF_SPERRANTRIEBIN.p_scInSperrAtRükOpen_fbiMaxErrorRetryAllowed)
    Image (10,52 32x32), invisible if: ITF_RückOffen_IN = 0, image: CtaVisSymbols.ImagePool.build
        OnMouseDown:  Dialog=SperrAntrieb_POPUP_IO_ITF, Parameters={ITF_IO_IN: ITF_RückOffen_IN}, OpenModal=True, OpenCentered=True
    Label (45,58 120x20), "IO- Konfiguration", invisible if: ITF_RückOffen_IN = 0
    Textfield (30,255 140x20), "%s", text list: 'CtaAppReport.txtLibAp99_2enTypeOfAck', text index: CtaSysConfig.fcGetEnumerationId(ITF_SPERRANTRIEBIN.p_scInSperrAtRükOpen_fbiTypeOfAck)
END_VISUALIZATION

// 40 Visualizations/POPUP/PARAMETER/SperrAntrieb_IO/SperrAntrieb_ParameterIO3
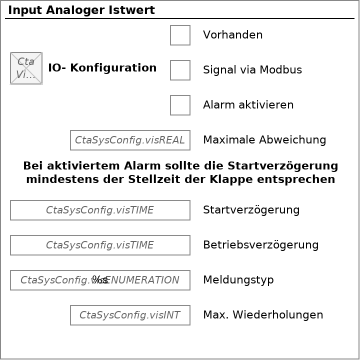
VISUALIZATION SperrAntrieb_ParameterIO3  // 360x360
VAR_INPUT
    ITF_SPERRANTRIEBIN 	:	ITF_SPERRANTRIEB;
	ITF_ActualPos_IN	:	CtaSysIO.ITF_IO;
END_VAR
    Label (5,0 350x20), "Input Analoger Istwert"
    Frame (170,25 20x20)
        shows CtaSysConfig.visBOOL(visfbBOOLIn := ITF_SPERRANTRIEBIN.p_scInSperrAtActualPosition_fbxEnable)
    Label (200,25 150x20), "Vorhanden"
    Frame (170,60 20x20)
        shows CtaSysConfig.visBOOL(visfbBOOLIn := ITF_SPERRANTRIEBIN.p_scInSperrAtActualPosition_fbxInputMb)
    Label (200,60 150x20), "Signal via Modbus"
    Frame (170,95 20x20)
        shows CtaSysConfig.visBOOL(visfbBOOLIn := ITF_SPERRANTRIEBIN.p_scInSperrAtActualPosition_fbxDoesAlarm)
    Label (200,95 150x20), "Alarm aktivieren"
    Frame (10,200 180x20)
        shows CtaSysConfig.visTIME(visfbTIMEIn := ITF_SPERRANTRIEBIN.p_scInSperrAtActualPosition_fbtDelayStart)
    Label (200,200 150x20), "Startverzögerung"
    Label (200,235 150x20), "Betriebsverzögerung"
    Frame (10,235 180x20)
        shows CtaSysConfig.visTIME(visfbTIMEIn := ITF_SPERRANTRIEBIN.p_scInSperrAtActualPosition_fbtDelayRun)
    Frame (70,130 120x20)
        shows CtaSysConfig.visREAL(visfbREALIn := ITF_SPERRANTRIEBIN.p_scInSperrAtActualPosition_fbrMaxDiff, stPhysikalischeEinheit := '%')
    Label (200,130 150x20), "Maximale Abweichung"
    Label (5,159 352x27), "Bei aktiviertem Alarm sollte die Startverzögerung mindestens der Stellzeit der Klappe entsprechen"
    Label (200,270 150x20), "Meldungstyp"
    Label (200,305 150x20), "Max. Wiederholungen"
    Line (5,18) (354,18)
    Frame (10,270 180x20)
        shows CtaSysConfig.visENUMERATION(visfbENUIn := ITF_SPERRANTRIEBIN.p_scInSperrAtActualPosition_fbiTypeOfAck)
    Frame (70,305 120x20)
        shows CtaSysConfig.visINT(visfbINTIn := ITF_SPERRANTRIEBIN.p_scInSperrAtActualPosition_fbiMaxErrorRetryAllowed)
    Image (10,52 32x32), invisible if: ITF_ActualPos_IN = 0, image: CtaVisSymbols.ImagePool.build
        OnMouseDown:  Dialog=SperrAntrieb_POPUP_IO_ITF, Parameters={ITF_IO_IN: ITF_ActualPos_IN}, OpenModal=True, OpenCentered=True
    Label (45,58 120x20), "IO- Konfiguration", invisible if: ITF_ActualPos_IN = 0
    Textfield (30,270 140x20), "%s", text list: 'CtaAppReport.txtLibAp99_2enTypeOfAck', text index: CtaSysConfig.fcGetEnumerationId(ITF_SPERRANTRIEBIN.p_scInSperrAtActualPosition_fbiTypeOfAck)
END_VISUALIZATION

// 40 Visualizations/POPUP/PARAMETER/SperrAntrieb_InfluxDb/SperrAntrieb_ParameterInfluxDb
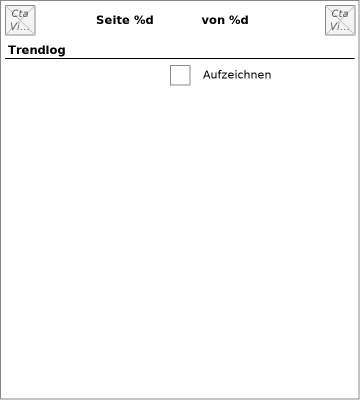
VISUALIZATION SperrAntrieb_ParameterInfluxDb  // 360x400
VAR_INPUT
    ITF_SPERRANTRIEBIN : ITF_SPERRANTRIEB;
END_VAR
VAR
    uiPage  :   UINT;
    uiMin   :   UINT    := 0;
    uiMax   :   UINT    := 0;
END_VAR
    Image (5,5 30x30), invisible if: uiPage = uiMin, image: CtaVisSymbols.ImagePool.arrow-left_square
        OnMouseClick: execute {
            uiPage := uiPage - 1;
            IF uiPage <= uiMin THEN
                uiPage := uiMin;
            END_IF;
        }
    Image (325,5 30x30), invisible if: uiPage = uiMax, image: CtaVisSymbols.ImagePool.arrow-right_square
        OnMouseClick: execute {
            uiPage := uiPage + 1;
            IF uiPage >= uiMax THEN
                uiPage := uiMax;
            END_IF;
        }
    Frame (0,40 360x360), frame switch variable: uiPage
        shows SperrAntrieb_ParameterInfluxDb0(ITF_SPERRANTRIEBIN := ITF_SPERRANTRIEBIN)
        shows AT_ParameterIO1(ITF_Parameter := ITF_Parameter)
        pReferences[0]: ITF_Parameter=ITF_Parameter
    Textfield (75,5 100x30), "Seite %d", text variable: uiPage
    Textfield (175,5 100x30), "von %d", text variable: uiMax
END_VISUALIZATION

// 40 Visualizations/POPUP/PARAMETER/SperrAntrieb_InfluxDb/SperrAntrieb_ParameterInfluxDb0
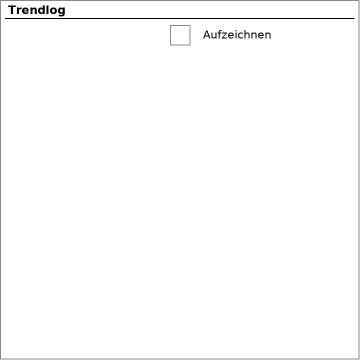
VISUALIZATION SperrAntrieb_ParameterInfluxDb0  // 360x360
VAR_INPUT
    ITF_SPERRANTRIEBIN : ITF_SPERRANTRIEB;
END_VAR
    Frame (170,25 20x20)
        shows CtaSysConfig.visBOOL(visfbBOOLIn := ITF_SPERRANTRIEBIN.p_scInfluxDb_fbxEnable)
    Label (200,25 150x20), "Aufzeichnen"
    Label (5,0 350x20), "Trendlog"
    Line (5,18) (354,18)
END_VISUALIZATION

// 40 Visualizations/POPUP/IO/SperrAntrieb_IO0
